// TIA Portal V19 export
FUNCTION "FC50_VacuumValve" : Void   // FC50, LAD
{ S7_Optimized_Access := 'TRUE' }
// stored: AutoNumber false, IsIECCheckEnabled true, SetENOAutomatically false
BEGIN

REGION Network 1: Manage Vacuum valve
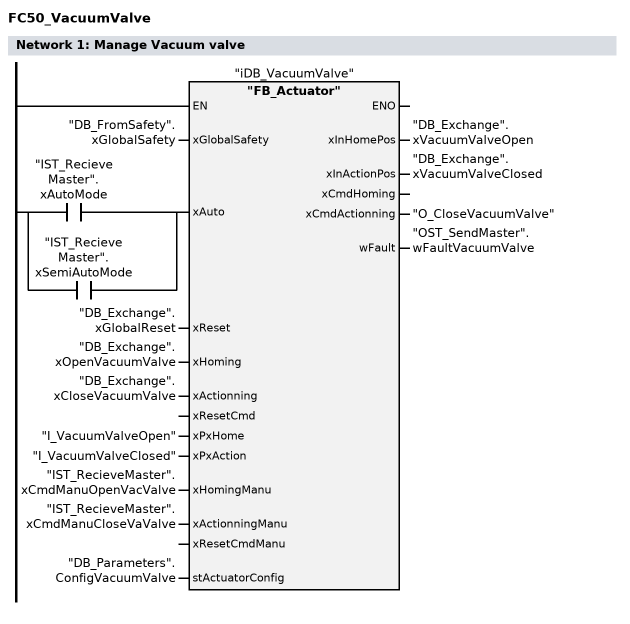
   RUNG wire#powerrail
      "iDB_VacuumValve"(xAuto := wire#w1, xGlobalSafety := "DB_FromSafety".xGlobalSafety, xReset := "DB_Exchange".xGlobalReset, xHoming := "DB_Exchange".xOpenVacuumValve, xActionning := "DB_Exchange".xCloseVacuumValve, xResetCmd :=, xPxHome := "I_VacuumValveOpen", xPxAction := "I_VacuumValveClosed", xHomingManu := "IST_RecieveMaster".xCmdManuOpenVacValve, xActionningManu := "IST_RecieveMaster".xCmdManuCloseVaValve, xResetCmdManu :=, stActuatorConfig := "DB_Parameters".ConfigVacuumValve, xInHomePos => "DB_Exchange".xVacuumValveOpen, xInActionPos => "DB_Exchange".xVacuumValveClosed, xCmdHoming =>, xCmdActionning => "O_CloseVacuumValve", wFault => "OST_SendMaster".wFaultVacuumValve)
   END_RUNG
   RUNG wire#powerrail
      Contact( "IST_RecieveMaster".xAutoMode )
   END_RUNG wire#w1
   RUNG wire#powerrail
      Contact( "IST_RecieveMaster".xSemiAutoMode )
   END_RUNG wire#w1
   // the same network as SCL:
   "iDB_VacuumValve"(xGlobalSafety := "DB_FromSafety".xGlobalSafety,   // "FB_Actuator"
                     xAuto := "IST_RecieveMaster".xAutoMode OR "IST_RecieveMaster".xSemiAutoMode,
                     xReset := "DB_Exchange".xGlobalReset,
                     xHoming := "DB_Exchange".xOpenVacuumValve,
                     xActionning := "DB_Exchange".xCloseVacuumValve,
                     xPxHome := "I_VacuumValveOpen",
                     xPxAction := "I_VacuumValveClosed",
                     xHomingManu := "IST_RecieveMaster".xCmdManuOpenVacValve,
                     xActionningManu := "IST_RecieveMaster".xCmdManuCloseVaValve,
                     stActuatorConfig := "DB_Parameters".ConfigVacuumValve,
                     xInHomePos => "DB_Exchange".xVacuumValveOpen,
                     xInActionPos => "DB_Exchange".xVacuumValveClosed,
                     xCmdActionning => "O_CloseVacuumValve",
                     wFault => "OST_SendMaster".wFaultVacuumValve);
END_REGION
END_FUNCTION
